INTERFACE I_LogSource EXTENDS I_Base

{attribute 'monitoring':='call'}
PROPERTY SourceName : T_MaxString
GET
END_GET
END_PROPERTY

{attribute 'monitoring':='call'}
PROPERTY Timestamp : T_FILETIME64
GET
END_GET
END_PROPERTY

END_INTERFACE

(* stored: Version 1.1.0.1, ProductVersion 3.1.4026.18
   Itf I_LogSource: Id {dfea656c-ea4c-46d2-a3c0-d9914a697ac9}
   Property SourceName: Id {eb0236da-b0f9-49dc-850f-464d21b1b8af}
   Get Get: Id {ee636fd3-ff5c-48db-9c13-856d5e9d938d}
   Property Timestamp: Id {ff7f8a0c-5fb9-455a-81d0-2dd92f9534eb}
   Get Get: Id {6d09911a-32ed-4386-b242-b9a8cfff859d} *)
